(* Schneider Machine Expert - Basic project motor_hours_tracking_TM221CE24T, file version 3.0.0.0 *)
(* ProjectInformations: Name=Motor Hours Tracking TM221CE24T *)

HARDWARE
  Cpu 0: TM221CE24T
  EthernetConfiguration: NetworkName=M221, IpAllocationMode=ByDhcp, IpAddress=192.168.1.10, SubnetMask=255.255.255.0
  SerialLineConfiguration: Baud=Baud19200, Parity=ParityEven, DataBits=DataBits8, StopBits=StopBits1, PhysicalMedium=PhysicalMediumRs485, TransmissionMode=TransmissionModeModbusRtu, SlaveId=1, Addressing=SlaveAddressing
  MastTask: UsePeriodScanMode=false, PeriodScan=100
  FastTask: Period=255
  CpuBehavior: StartingMode=StartAsPreviousState, AutoSaveRamOnEeprom=true, WatchdogPeriod=250

SYMBOLS  (address, symbol, comment, settings)
  %M0       MTR_RUN  "Motor running latch"
  %M1       MAINT_REQ  "Maintenance required flag (100 hours reached)"
  %C0         [Preset=6000]
  %I0.0     PB_START
  %I0.1     PB_STOP
  %I0.2     ESTOP
  %I0.3     PB_MAINT_RST
  %Q0.0     MTR_CONTACTOR
  %Q0.1     LT_RUN
  %Q0.2     LT_MAINT

POU Motor Hours Tracking
  (* SectionNumber=1 *)

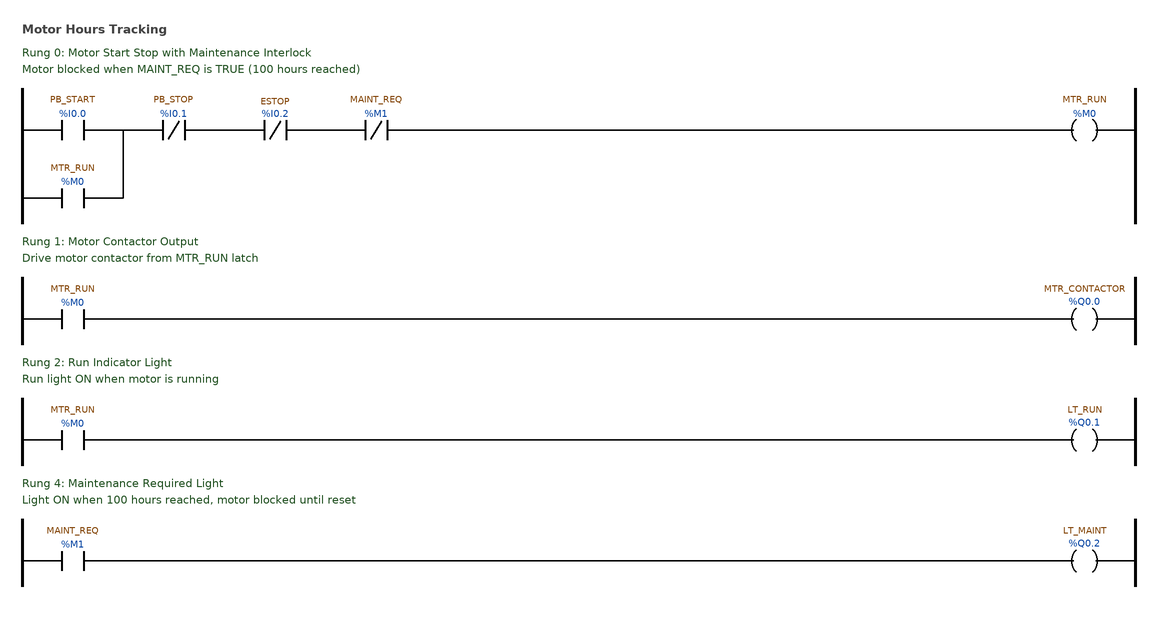

// Rung 0: Motor Start Stop with Maintenance Interlock
// Motor blocked when MAINT_REQ is TRUE (100 hours reached)
  LD %I0.0                (* PB_START *)
  OR %M0                  (* MTR_RUN *)
  ANDN %I0.1              (* PB_STOP *)
  ANDN %I0.2              (* ESTOP *)
  ANDN %M1                (* MAINT_REQ *)
  ST %M0                  (* MTR_RUN *)
  // as ST:
  //   MTR_RUN := (PB_START OR MTR_RUN) AND NOT PB_STOP AND NOT ESTOP AND NOT MAINT_REQ;

// Rung 1: Motor Contactor Output
// Drive motor contactor from MTR_RUN latch
  LD %M0                  (* MTR_RUN *)
  ST %Q0.0                (* MTR_CONTACTOR *)
  // as ST:
  //   MTR_CONTACTOR := MTR_RUN;

// Rung 2: Run Indicator Light
// Run light ON when motor is running
  LD %M0                  (* MTR_RUN *)
  ST %Q0.1                (* LT_RUN *)
  // as ST:
  //   LT_RUN := MTR_RUN;

// Rung 3: Minutes Counter with Reset
// Row 0: R input (reset). Row 2: CU input (MTR_RUN AND %S7). Preset 6000 = 100 hours
  BLK %C0
  LD %I0.3                (* PB_MAINT_RST *)
  R
  LD %M0                  (* MTR_RUN *)
  AND %S7
  CU
  OUT_BLK
  LD D
  ST %M1                  (* MAINT_REQ *)
  END_BLK
  // as ST:
  //   %C0(R := PB_MAINT_RST, CU := MTR_RUN AND %S7);
  //   MAINT_REQ := %C0.D;
  (* the ladder stored for this rung does not match its IL; not drawn *)

// Rung 4: Maintenance Required Light
// Light ON when 100 hours reached, motor blocked until reset
  LD %M1                  (* MAINT_REQ *)
  ST %Q0.2                (* LT_MAINT *)
  // as ST:
  //   LT_MAINT := MAINT_REQ;
